TYPE Dense_v1_LayerWeights:
STRUCT
    normalization_mean : ARRAY[0..0] OF LREAL;
    normalization_std : ARRAY[0..0] OF LREAL;
    HiddenLayers1_weight : ARRAY[0..3,0..2] OF LREAL;
    HiddenLayers1_bias : ARRAY[0..3] OF LREAL;
    HiddenLayers2_weight : ARRAY[0..4,0..3] OF LREAL;
    HiddenLayers2_bias : ARRAY[0..4] OF LREAL;
    HiddenLayers3_weight : ARRAY[0..5,0..4] OF LREAL;
    HiddenLayers3_bias : ARRAY[0..5] OF LREAL;
    OutputLayer_weight : ARRAY[0..0,0..5] OF LREAL;
    OutputLayer_bias : ARRAY[0..0] OF LREAL;
    denormalization_mean : ARRAY[0..0] OF LREAL;
    denormalization_std : ARRAY[0..0] OF LREAL;
    
END_STRUCT
END_TYPE

(* stored: Version 1.1.0.1, ProductVersion 3.1.4024.12
   DUT Dense_v1_LayerWeights: Id {4cce5101-8a01-4105-95e3-5a33056e8af0} *)
